// TIA Portal project "babu_3MotorsUsingComparators" (V15)

(* hardware
DEVICE "S7-1200 station_1"  S7-1200 Station
   slot 0: "Rack_0"  S7-1200 Rack  Rack  V1.0
   slot 1: "PLC_1"  CPU 1212C DC/DC/DC  6ES7 212-1AE40-0XB0  V4.2
*)

// ===== PLC "PLC_1"  CPU 1212C DC/DC/DC =====

VAR_GLOBAL   // PLC tag table "Default tag table"
   "INPUT" AT %M0.0 : Bool;
   "POSITIVE SIGNAL" AT %M0.1 : Bool;
   "IN OUT" AT %M0.2 : Bool;
   "OUTPUT" AT %Q0.0 : Bool;
   "IP2" AT %M0.3 : Bool;
   "OP2" AT %Q0.1 : Bool;
   "OP21" AT %Q0.2 : Bool;
   "IP3" AT %M0.4 : Bool;
   "OP3" AT %M0.5 : Bool;
   "OP31" AT %Q0.3 : Bool;
   "POWER ON MEM" AT %M0.6 : Bool;
   "POWER ON" AT %M0.7 : Bool;
   "CYCLE COMPLETE" AT %M1.0 : Bool;
   "RESET" AT %M1.1 : Bool;
   "MOTOR1" AT %Q0.4 : Bool;
   "MOTOR2" AT %Q0.5 : Bool;
   "MOTOR3" AT %Q0.6 : Bool;
   "MEM1" AT %M1.2 : Bool;
   "MEM2" AT %M1.3 : Bool;
END_VAR

// folder: System blocks/Program resources

DATA_BLOCK "IEC_Counter_0_DB"   // DB1
{ S7_Optimized_Access := 'TRUE' }
AUTHOR : Simatic
FAMILY : IEC
NAME : CNTR
VERSION : 1.0
// stored: InstanceOfName IEC_COUNTER
"IEC_COUNTER"
BEGIN
END_DATA_BLOCK

DATA_BLOCK "IEC_Counter_0_DB_1"   // DB2
{ S7_Optimized_Access := 'TRUE' }
AUTHOR : Simatic
FAMILY : IEC
NAME : CNTR
VERSION : 1.0
// stored: InstanceOfName IEC_COUNTER
"IEC_COUNTER"
BEGIN
END_DATA_BLOCK

DATA_BLOCK "IEC_Timer_0_DB"   // DB3
{ S7_Optimized_Access := 'TRUE' }
AUTHOR : Simatic
FAMILY : IEC
NAME : IEC_TMR
VERSION : 1.0
// stored: InstanceOfName IEC_TIMER
"IEC_TIMER"
BEGIN
END_DATA_BLOCK

DATA_BLOCK "IEC_Timer_0_DB_1"   // DB4
{ S7_Optimized_Access := 'TRUE' }
AUTHOR : Simatic
FAMILY : IEC
NAME : IEC_TMR
VERSION : 1.0
// stored: InstanceOfName IEC_TIMER
"IEC_TIMER"
BEGIN
END_DATA_BLOCK

// folder: (top level)

ORGANIZATION_BLOCK "Main"   // OB1, LAD, ProgramCycle
TITLE = "Main Program Sweep (Cycle)"
{ S7_Optimized_Access := 'TRUE' }
VERSION : 0.1
   VAR_INPUT
      Initial_Call : Bool;   // Initial call of this OB
      Remanence : Bool;   // =True, if remanent data are available
   END_VAR
   VAR_TEMP   // added for the SCL form of the ladder/FBD networks
      _w1 : Bool;
   END_VAR
BEGIN

REGION Network 1
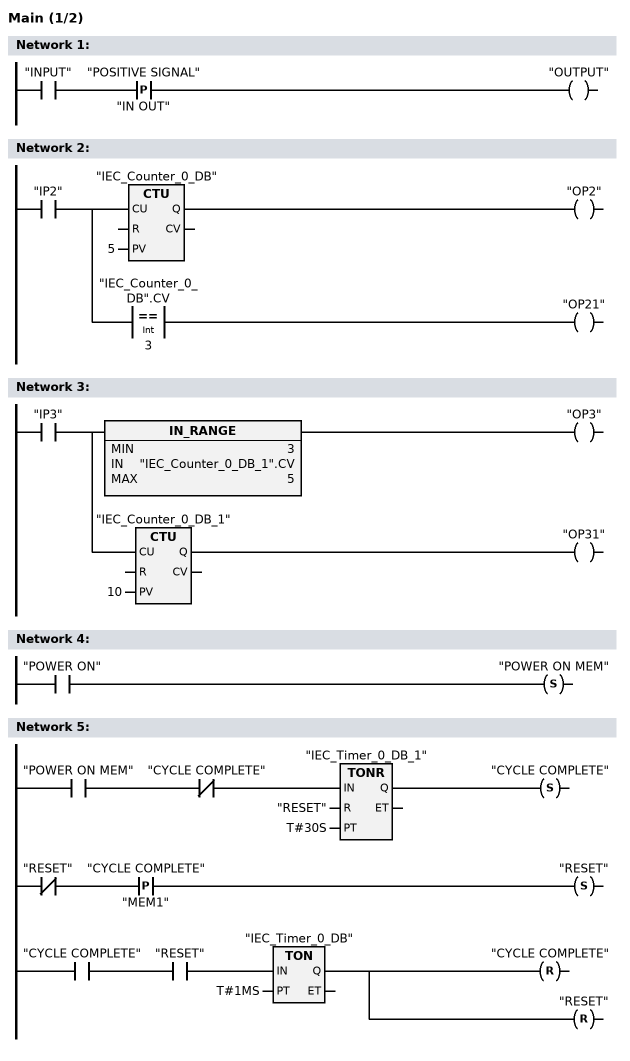
   RUNG wire#powerrail
      Contact( "INPUT" )
      P_Contact(operand := "POSITIVE SIGNAL", bit := "IN OUT")
      Coil( "OUTPUT" )
   END_RUNG
   // the same network as SCL:
   #_w1 := "INPUT" AND "POSITIVE SIGNAL" AND NOT "IN OUT";   // rising edge of "POSITIVE SIGNAL"
   "IN OUT" := "POSITIVE SIGNAL";
   "OUTPUT" := #_w1;
END_REGION

REGION Network 2
   "IEC_Counter_0_DB".CTU(CU := "IP2", PV := 5);
   "OP2" := "IEC_Counter_0_DB".Q;
   "OP21" := "IP2" AND ("IEC_Counter_0_DB".CV = 3);
END_REGION

REGION Network 3
   "OP3" := "IP3" AND (3 <= "IEC_Counter_0_DB_1".CV) AND ("IEC_Counter_0_DB_1".CV <= 5);
   "IEC_Counter_0_DB_1".CTU(CU := "IP3", PV := 10);
   "OP31" := "IEC_Counter_0_DB_1".Q;
END_REGION

REGION Network 4
   RUNG wire#powerrail
      Contact( "POWER ON" )
      S_Coil( "POWER ON MEM" )
   END_RUNG
   // the same network as SCL:
   IF "POWER ON" THEN "POWER ON MEM" := TRUE; END_IF;
END_REGION

REGION Network 5
   "IEC_Timer_0_DB_1".TONR(IN := "POWER ON MEM" AND NOT "CYCLE COMPLETE", R := "RESET", PT := T#30S);
   IF "IEC_Timer_0_DB_1".Q THEN "CYCLE COMPLETE" := TRUE; END_IF;
   #_w1 := NOT "RESET" AND "CYCLE COMPLETE" AND NOT "MEM1";   // rising edge of "CYCLE COMPLETE"
   "MEM1" := "CYCLE COMPLETE";
   IF #_w1 THEN "RESET" := TRUE; END_IF;
   "IEC_Timer_0_DB".TON(IN := "CYCLE COMPLETE" AND "RESET", PT := T#1MS);
   IF "IEC_Timer_0_DB".Q THEN
       "CYCLE COMPLETE" := FALSE;
       "RESET" := FALSE;
   END_IF;
END_REGION

REGION Network 6
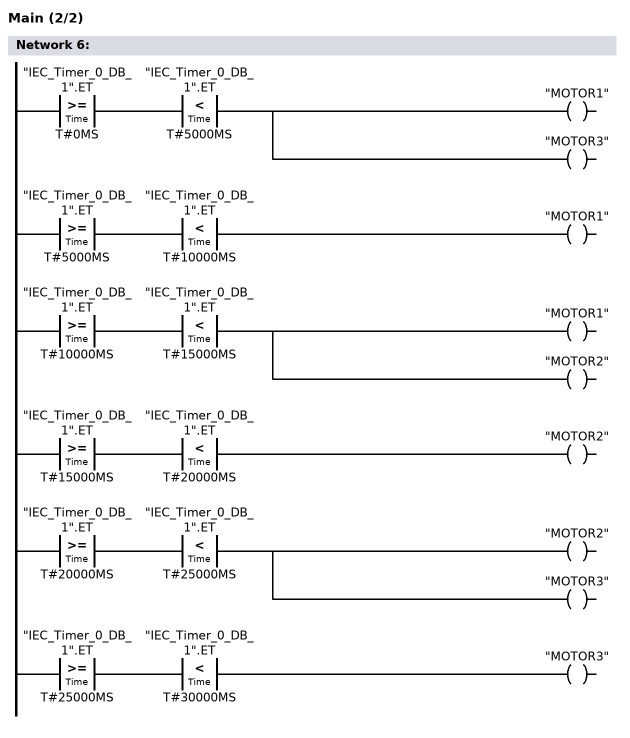
   RUNG wire#powerrail
      { S7_Templates := "SrcType := Time" } GE_Contact(in1 := "IEC_Timer_0_DB_1".ET, in2 := T#0MS)
      { S7_Templates := "SrcType := Time" } LT_Contact(in1 := "IEC_Timer_0_DB_1".ET, in2 := T#5000MS)
      wire#w1
      Coil( "MOTOR1" )
   END_RUNG
   RUNG wire#w1
      Coil( "MOTOR3" )
   END_RUNG
   RUNG wire#powerrail
      { S7_Templates := "SrcType := Time" } GE_Contact(in1 := "IEC_Timer_0_DB_1".ET, in2 := T#5000MS)
      { S7_Templates := "SrcType := Time" } LT_Contact(in1 := "IEC_Timer_0_DB_1".ET, in2 := T#10000MS)
      Coil( "MOTOR1" )
   END_RUNG
   RUNG wire#powerrail
      { S7_Templates := "SrcType := Time" } GE_Contact(in1 := "IEC_Timer_0_DB_1".ET, in2 := T#10000MS)
      { S7_Templates := "SrcType := Time" } LT_Contact(in1 := "IEC_Timer_0_DB_1".ET, in2 := T#15000MS)
      wire#w2
      Coil( "MOTOR1" )
   END_RUNG
   RUNG wire#w2
      Coil( "MOTOR2" )
   END_RUNG
   RUNG wire#powerrail
      { S7_Templates := "SrcType := Time" } GE_Contact(in1 := "IEC_Timer_0_DB_1".ET, in2 := T#15000MS)
      { S7_Templates := "SrcType := Time" } LT_Contact(in1 := "IEC_Timer_0_DB_1".ET, in2 := T#20000MS)
      Coil( "MOTOR2" )
   END_RUNG
   RUNG wire#powerrail
      { S7_Templates := "SrcType := Time" } GE_Contact(in1 := "IEC_Timer_0_DB_1".ET, in2 := T#20000MS)
      { S7_Templates := "SrcType := Time" } LT_Contact(in1 := "IEC_Timer_0_DB_1".ET, in2 := T#25000MS)
      wire#w3
      Coil( "MOTOR2" )
   END_RUNG
   RUNG wire#w3
      Coil( "MOTOR3" )
   END_RUNG
   RUNG wire#powerrail
      { S7_Templates := "SrcType := Time" } GE_Contact(in1 := "IEC_Timer_0_DB_1".ET, in2 := T#25000MS)
      { S7_Templates := "SrcType := Time" } LT_Contact(in1 := "IEC_Timer_0_DB_1".ET, in2 := T#30000MS)
      Coil( "MOTOR3" )
   END_RUNG
   // the same network as SCL:
   "MOTOR1" := ("IEC_Timer_0_DB_1".ET >= T#0MS) AND ("IEC_Timer_0_DB_1".ET < T#5000MS);
   "MOTOR3" := "MOTOR1";
   "MOTOR1" := ("IEC_Timer_0_DB_1".ET >= T#5000MS) AND ("IEC_Timer_0_DB_1".ET < T#10000MS);
   "MOTOR1" := ("IEC_Timer_0_DB_1".ET >= T#10000MS) AND ("IEC_Timer_0_DB_1".ET < T#15000MS);
   "MOTOR2" := "MOTOR1";
   "MOTOR2" := ("IEC_Timer_0_DB_1".ET >= T#15000MS) AND ("IEC_Timer_0_DB_1".ET < T#20000MS);
   "MOTOR2" := ("IEC_Timer_0_DB_1".ET >= T#20000MS) AND ("IEC_Timer_0_DB_1".ET < T#25000MS);
   "MOTOR3" := "MOTOR2";
   "MOTOR3" := ("IEC_Timer_0_DB_1".ET >= T#25000MS) AND ("IEC_Timer_0_DB_1".ET < T#30000MS);
END_REGION
END_ORGANIZATION_BLOCK